TYPE "PLCtoMES_MainCheckOut_ext"
VERSION : 0.1
   STRUCT
      Unload_Station1DataSaveReq : Bool;
      Unload_Station2DataSaveReq : Bool;
      Unload_Station3DataSaveReq : Bool;
      Unload_Station4DataSaveReq : Bool;
      Unload_Station5DataSaveReq : Bool;
      Unload_Station6DataSaveReq : Bool;
      Unload_Station7DataSaveReq : Bool;
      Unload_Station8DataSaveReq : Bool;
   END_STRUCT;

END_TYPE

